FUNCTION_BLOCK Atuador_Coester_CSR6T (* Composite Function Block Type *)
  (* Standard: 61499-2 *)
  (* Version 0.0, 1/26/2026, Schneider Electric, template *)
  PACKAGE Hidryco.HidrycoLib;
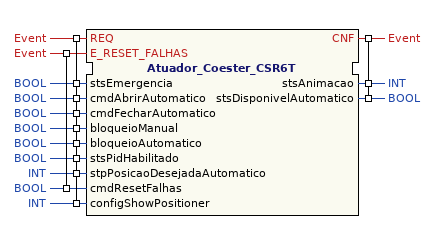
  EVENT_INPUT
    REQ WITH cmdAbrirAutomatico, cmdFecharAutomatico, bloqueioManual, bloqueioAutomatico, stsPidHabilitado, stpPosicaoDesejadaAutomatico, configShowPositioner, stsEmergencia;
    E_RESET_FALHAS WITH cmdResetFalhas;
  END_EVENT
  EVENT_OUTPUT
    CNF WITH stsAnimacao, stsDisponivelAutomatico;
  END_EVENT
  VAR_INPUT
    stsEmergencia : BOOL;
    cmdAbrirAutomatico : BOOL;
    cmdFecharAutomatico : BOOL;
    bloqueioManual : BOOL;
    bloqueioAutomatico : BOOL;
    stsPidHabilitado : BOOL;
    stpPosicaoDesejadaAutomatico : INT; (* Saida do PID *)
    cmdResetFalhas : BOOL;
    configShowPositioner : INT; (* Alterar a porcentagem de abertura (0 - Only ON OFF, 1 - With Positioner) *)
  END_VAR
  VAR_OUTPUT
    stsAnimacao : INT;
    stsDisponivelAutomatico : BOOL;
  END_VAR
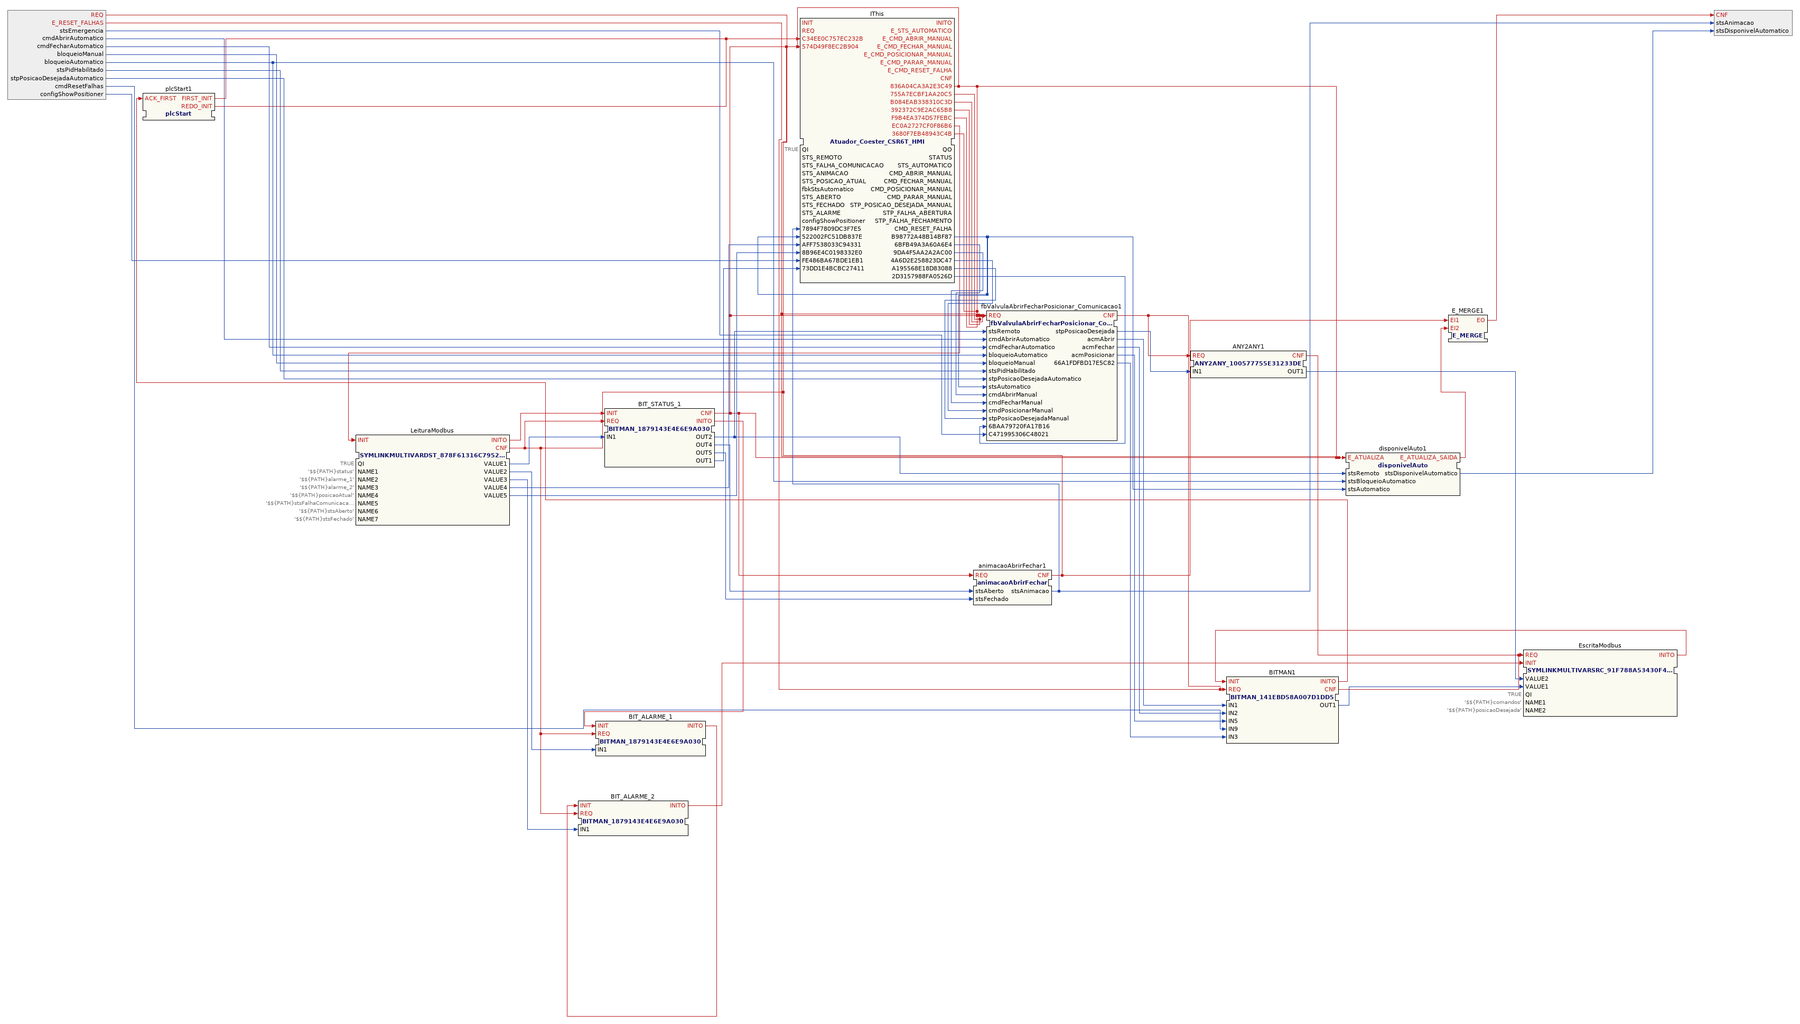
  (* Bits de status 1: 0 modo de operação local 1 modo de operação remoto 2 modo de operação desligado 3 posição aberta 4 posição fechada 5 posição intermediária 6 movimento de abertura 7 movimento de fechamento 8 atuador(válvula) parado 9 motor energizado 10 movimento manual 11 aberto com torque 12 fechado com torque 13 modo Modbus *)
  (* Bits de Alarme 1: 0 modo de operação não remoto 1 parada local de emergência 2 parada antecipada por torque na abertura 3 parada antecipada por torque no fechamento 4 atuador(válvula) travado 5 operação incompleta 6 sobreaquecimento do motor 7 falha no motor ao energizar 8 motor energizado após fim de curso 9 motor energizado após comando de parada 10 falha de comando 11 falta de fase 12 atuador não programado *)
  (* Bits de Alarme 2: 0 tensão de alimentação alta 1 tensão de alimentação baixa 2 tensão de bateria baixa 3 4 fim de curso mecânico ultrapassado na abertura 5 fim de curso mecânico ultrapassado no fechamento 6 fim de curso programado ultrapassado na abertura 7 fim de curso programado ultrapassado no fechamento 8 cartão anybus não detectado *)
  (* Bits de comando 0 abrir 1 fechar 2 parar 3 ESD 4 posicionar 5 PST (Partial Stroke Test) 6 espera 7 espera 8 quitar alarmes *)
  FBS
    IThis : Atuador_Coester_CSR6T_HMI(QI := TRUE);
    LeituraModbus : SYMLINKMULTIVARDST_878F61316C795212(QI := TRUE, NAME1 := '$${PATH}status', NAME2 := '$${PATH}alarme_1', NAME3 := '$${PATH}alarme_2', NAME4 := '$${PATH}posicaoAtual', NAME5 := '$${PATH}stsFalhaComunicacao', NAME6 := '$${PATH}stsAberto', NAME7 := '$${PATH}stsFechado'); {SET_ATTRIBUTE(Configuration.GenericFBType.InterfaceParams, Runtime.System#I:=7;VALUE${I$}:WORD,WORD,WORD,INT,BOOL,BOOL,BOOL)}
    plcStart1 : plcStart;
    EscritaModbus : SYMLINKMULTIVARSRC_91F788A53430F44E(QI := TRUE, NAME1 := '$${PATH}comandos', NAME2 := '$${PATH}posicaoDesejada'); {SET_ATTRIBUTE(Configuration.GenericFBType.InterfaceParams, Runtime.System#I:=2;VALUE${I$}:WORD,WORD)}
    BITMAN1 : BITMAN_141EBD58A007D1DD5; {SET_ATTRIBUTE(Configuration.GenericFBType.InterfaceParams, Runtime.Standard#CNTIN:=9;CNTOUT:=1;IN${CNTIN$}:BOOL,BOOL,BOOL,BOOL,BOOL,BOOL,BOOL,BOOL,BOOL;OUT${CNTOUT$}:WORD)}
    BIT_STATUS_1 : BITMAN_1879143E4E6E9A030; {SET_ATTRIBUTE(Configuration.GenericFBType.InterfaceParams, Runtime.Standard#CNTIN:=1;CNTOUT:=16;IN${CNTIN$}:WORD;OUT${CNTOUT$}:BOOL,BOOL,BOOL,BOOL,BOOL,BOOL,BOOL,BOOL,BOOL,BOOL,BOOL,BOOL,BOOL,BOOL,BOOL,BOOL)}
    BIT_ALARME_1 : BITMAN_1879143E4E6E9A030; {SET_ATTRIBUTE(Configuration.GenericFBType.InterfaceParams, Runtime.Standard#CNTIN:=1;CNTOUT:=16;IN${CNTIN$}:WORD;OUT${CNTOUT$}:BOOL,BOOL,BOOL,BOOL,BOOL,BOOL,BOOL,BOOL,BOOL,BOOL,BOOL,BOOL,BOOL,BOOL,BOOL,BOOL)}
    BIT_ALARME_2 : BITMAN_1879143E4E6E9A030; {SET_ATTRIBUTE(Configuration.GenericFBType.InterfaceParams, Runtime.Standard#CNTIN:=1;CNTOUT:=16;IN${CNTIN$}:WORD;OUT${CNTOUT$}:BOOL,BOOL,BOOL,BOOL,BOOL,BOOL,BOOL,BOOL,BOOL,BOOL,BOOL,BOOL,BOOL,BOOL,BOOL,BOOL)}
    fbValvulaAbrirFecharPosicionar_Comunicacao1 : fbValvulaAbrirFecharPosicionar_Comunicacao;
    animacaoAbrirFechar1 : animacaoAbrirFechar;
    ANY2ANY1 : ANY2ANY_100577755E31233DE; {SET_ATTRIBUTE(Configuration.GenericFBType.InterfaceParams, Runtime.Standard#CNT:=1;IN${CNT$}:INT;OUT${CNT$}:WORD)}
    disponivelAuto1 : disponivelAuto; {SET_ATTRIBUTE(Configuration.Component.HideUnusedPorts, )}
    E_MERGE1 : E_MERGE;
  END_FBS
  EVENT_CONNECTIONS
    fbValvulaAbrirFecharPosicionar_Comunicacao1.CNF TO ANY2ANY1.REQ;
    ANY2ANY1.CNF TO EscritaModbus.REQ;
    BIT_STATUS_1.CNF TO fbValvulaAbrirFecharPosicionar_Comunicacao1.REQ;
    BIT_STATUS_1.CNF TO animacaoAbrirFechar1.REQ;
    REQ TO fbValvulaAbrirFecharPosicionar_Comunicacao1.REQ;
    BIT_STATUS_1.INITO TO BIT_ALARME_1.INIT;
    BIT_ALARME_1.INITO TO BIT_ALARME_2.INIT;
    BIT_ALARME_2.INITO TO EscritaModbus.INIT;
    animacaoAbrirFechar1.CNF TO E_MERGE1.EI1;
    BIT_STATUS_1.CNF TO disponivelAuto1.E_ATUALIZA;
    REQ TO disponivelAuto1.E_ATUALIZA;
    disponivelAuto1.E_ATUALIZA_SAIDA TO E_MERGE1.EI2;
    E_MERGE1.EO TO CNF;
    EscritaModbus.INITO TO BITMAN1.INIT;
    BITMAN1.INITO TO plcStart1.ACK_FIRST;
    E_RESET_FALHAS TO BITMAN1.REQ;
    BITMAN1.CNF TO EscritaModbus.REQ;
    fbValvulaAbrirFecharPosicionar_Comunicacao1.CNF TO BITMAN1.REQ;
    plcStart1.FIRST_INIT TO IThis.C34EE0C757EC232B;
    plcStart1.REDO_INIT TO IThis.C34EE0C757EC232B;
    BIT_STATUS_1.CNF TO IThis.574D49F8EC2B904;
    animacaoAbrirFechar1.CNF TO IThis.574D49F8EC2B904;
    IThis.836A04CA3A2E3C49 TO fbValvulaAbrirFecharPosicionar_Comunicacao1.REQ;
    IThis.836A04CA3A2E3C49 TO disponivelAuto1.E_ATUALIZA;
    IThis.755A7ECBF1AA20C5 TO fbValvulaAbrirFecharPosicionar_Comunicacao1.REQ;
    IThis.B084EAB338310C3D TO fbValvulaAbrirFecharPosicionar_Comunicacao1.REQ;
    IThis.392372C9E2AC65B8 TO fbValvulaAbrirFecharPosicionar_Comunicacao1.REQ;
    IThis.F9B4EA374D57FEBC TO fbValvulaAbrirFecharPosicionar_Comunicacao1.REQ;
    IThis.836A04CA3A2E3C49 TO IThis.574D49F8EC2B904;
    IThis.EC0A2727CF0F86B6 TO LeituraModbus.INIT;
    LeituraModbus.INITO TO BIT_STATUS_1.INIT;
    LeituraModbus.CNF TO BIT_STATUS_1.REQ;
    LeituraModbus.CNF TO BIT_ALARME_1.REQ;
    LeituraModbus.CNF TO BIT_ALARME_2.REQ;
    LeituraModbus.CNF TO IThis.574D49F8EC2B904;
    IThis.3680F7EB48943C4B TO fbValvulaAbrirFecharPosicionar_Comunicacao1.REQ;
  END_CONNECTIONS
  DATA_CONNECTIONS
    BIT_STATUS_1.OUT2 TO fbValvulaAbrirFecharPosicionar_Comunicacao1.stsRemoto;
    BIT_STATUS_1.OUT4 TO animacaoAbrirFechar1.stsAberto;
    BIT_STATUS_1.OUT5 TO animacaoAbrirFechar1.stsFechado;
    fbValvulaAbrirFecharPosicionar_Comunicacao1.stpPosicaoDesejada TO ANY2ANY1.IN1;
    ANY2ANY1.OUT1 TO EscritaModbus.VALUE2;
    cmdAbrirAutomatico TO fbValvulaAbrirFecharPosicionar_Comunicacao1.cmdAbrirAutomatico;
    cmdFecharAutomatico TO fbValvulaAbrirFecharPosicionar_Comunicacao1.cmdFecharAutomatico;
    bloqueioAutomatico TO fbValvulaAbrirFecharPosicionar_Comunicacao1.bloqueioAutomatico;
    bloqueioManual TO fbValvulaAbrirFecharPosicionar_Comunicacao1.bloqueioManual;
    stsPidHabilitado TO fbValvulaAbrirFecharPosicionar_Comunicacao1.stsPidHabilitado;
    stpPosicaoDesejadaAutomatico TO fbValvulaAbrirFecharPosicionar_Comunicacao1.stpPosicaoDesejadaAutomatico;
    animacaoAbrirFechar1.stsAnimacao TO stsAnimacao;
    BIT_STATUS_1.OUT2 TO disponivelAuto1.stsRemoto;
    bloqueioAutomatico TO disponivelAuto1.stsBloqueioAutomatico;
    disponivelAuto1.stsDisponivelAutomatico TO stsDisponivelAutomatico;
    fbValvulaAbrirFecharPosicionar_Comunicacao1.acmAbrir TO BITMAN1.IN1;
    fbValvulaAbrirFecharPosicionar_Comunicacao1.acmFechar TO BITMAN1.IN2;
    fbValvulaAbrirFecharPosicionar_Comunicacao1.acmPosicionar TO BITMAN1.IN5;
    BITMAN1.OUT1 TO EscritaModbus.VALUE1;
    cmdResetFalhas TO BITMAN1.IN9;
    animacaoAbrirFechar1.stsAnimacao TO IThis.7894F7809DC3F7E5;
    IThis.B98772A48B14BF87 TO IThis.522002FC51DB837E;
    IThis.B98772A48B14BF87 TO fbValvulaAbrirFecharPosicionar_Comunicacao1.stsAutomatico;
    IThis.B98772A48B14BF87 TO disponivelAuto1.stsAutomatico;
    IThis.6BFB49A3A60A6E4 TO fbValvulaAbrirFecharPosicionar_Comunicacao1.cmdAbrirManual;
    IThis.9DA4F5AA2A2AC00 TO fbValvulaAbrirFecharPosicionar_Comunicacao1.cmdFecharManual;
    IThis.4A6D2E258823DC47 TO fbValvulaAbrirFecharPosicionar_Comunicacao1.cmdPosicionarManual;
    IThis.A195568E18D83088 TO fbValvulaAbrirFecharPosicionar_Comunicacao1.stpPosicaoDesejadaManual;
    LeituraModbus.VALUE1 TO BIT_STATUS_1.IN1;
    LeituraModbus.VALUE2 TO BIT_ALARME_1.IN1;
    LeituraModbus.VALUE3 TO BIT_ALARME_2.IN1;
    LeituraModbus.VALUE4 TO IThis.AFF7538033C94331;
    LeituraModbus.VALUE5 TO IThis.8B96E4C0198332E0;
    configShowPositioner TO IThis.FE486BA67BDE1EB1;
    IThis.2D3157988FA0526D TO fbValvulaAbrirFecharPosicionar_Comunicacao1.6BAA79720FA17B16;
    fbValvulaAbrirFecharPosicionar_Comunicacao1.66A1FDFBD17E5C82 TO BITMAN1.IN3;
    stsEmergencia TO fbValvulaAbrirFecharPosicionar_Comunicacao1.C471995306C48021;
    BIT_STATUS_1.OUT1 TO IThis.73DD1E4BCBC27411;
  END_CONNECTIONS
END_FUNCTION_BLOCK
